Fanuc KAREL source: kt00598.KL

-- PROVISIONAL review KL for V940-1; original PC SHA256 7f11bc65f270600e1cfc9e00304e44312fb03ffb0b5b4f7e3eab36b4a6ac41e1
-- Incomplete behavior may be omitted. Consult companion uncertainty JSON. Do not deploy.
PROGRAM KT00598
%NOLOCKGROUP
VAR
  I1 : INTEGER
  I2 : INTEGER
  OUT : INTEGER
BEGIN
  -- V9_ZERO_TABLE_METADATA_HINT layout=0001; no indexed target words; source/name/runtime held
  -- UNRESOLVED_PC offsets 5-16; opcodes 2E,23
  -- UNRESOLVED_PC offsets 21-32; opcodes 2E,23
  -- UNRESOLVED_PC offsets 37-48; opcodes 2E,23
  -- UNRESOLVED_PC offsets 53-64; opcodes 2E,23
  -- UNRESOLVED_PC offsets 69-82; opcodes 21,48,23
  -- UNRESOLVED_PC offsets 87-91; opcodes 7F
END KT00598
